Yaskawa INFORM job: UPDATE_UF.JBI

/JOB
//NAME UPDATE_UF
///FOLDERNAME FOLDER001
//POS
///NPOS 2,0,0,2,0,0
///TOOL 1
///POSTYPE PULSE
///PULSE
C00000=-652,-17775,21844,-416,-82513,491
C00001=-361,56948,97542,-215,-89436,245
///POSTYPE ROBOT
///RECTAN
///RCONF 1,0,0,0,0,0,0,0,0,0,0,0,0,0,0,0,0,0,0,0,0,0,0,0
P00124=792.896,161.791,493.972,179.9986,-9.9993,0.0008
P00126=792.896,260.291,501.972,179.9986,-9.9993,0.0008
//INST
///DATE 2025/09/30 15:51
///ATTR SC,RW
///GROUP1 RB1
///LVARS 0,0,10,0,0,0,0,0
NOP
SFTOF
JUMP *LABEL
MOVL C00000 V=166.7
MOVL C00001 V=166.7
*LABEL
GETPOS PX124 STEP#(1)
GETPOS PX125 STEP#(2)
CNVRT PX124 PX124 RF
CNVRT PX125 PX125 RF
SET P126 P124
GETE D098 P124 (2)
ADD D098 100000
SETE P126 (2) D098
MFRAME UF#(15) PX124 PX125 PX126
END
